FUNCTION_BLOCK FB_Moving_average
VAR_INPUT
	New_sample: REAL;
	Num_samples: INT;
END_VAR
VAR_OUTPUT
	Out: REAL;
END_VAR
VAR CONSTANT
	Array_size: INT := 300;	
END_VAR
VAR
	Samples: ARRAY[0..(Array_size - 1)] OF REAL;
	i: INT;
	Sum: REAL;
	Pulse: BOOL;
	Toggle: BOOL;
END_VAR

(* Shift all the array elements one position and add them up while doing so *)
Sum:= 0;
FOR i:= 1 TO Num_samples - 1 DO
	Samples[Num_samples - i]:= Samples[Num_samples - i - 1];
	Sum:= Sum + Samples[Num_samples - i];
END_FOR

(* Insert the new sample into the array and add it to the sum *)
Samples[0]:= New_sample;
Sum:= Sum + New_sample;

(* Calculate the average *)
Out:= Sum / INT_TO_REAL(Num_samples);

END_FUNCTION_BLOCK

(* stored: Version 1.1.0.1, ProductVersion 3.1.4024.0
   POU FB_Moving_average: Id {cc1678d2-24a6-4224-94e3-0f7b70532a0d}, SpecialFunc None *)
